FUNCTION_BLOCK FB_System_BelHa
VAR_INPUT
	Freigabe_auto			: BOOL:=TRUE;
	Betrieb_Anford_auto		: BOOL:=TRUE;
	Regelung_Sollw_auto		: REAL;
	AdressType				: E_DALIV2AddrType;
END_VAR
VAR_OUTPUT
	{attribute 'OPC.UA.DA' := '1'}Steuerung				: ST_System_Bel_Steuerung;		
	{attribute 'OPC.UA.DA' := '1'}Stellwert				: ST_System_Bel_Stellwert;		
	{attribute 'OPC.UA.DA' := '1'}Zustand					: ST_System_Bel_Zustand;	
	{attribute 'OPC.UA.DA' := '1'}Parameter				: ST_System_Bel_Parameter;		
	Parameter_Regelung		: ST_Bel_Parameter;
	Parameter_Filter		: ST_Bel_Parameter;
END_VAR
VAR
	Ablaufsteuerung			: FB_System_BelHa_Ablaufsteuerung;
	Zustandscheck			: FB_System_BelHa_Zustandscheck;
	Logik 					: FB_System_BelHa_Logik;
	Sollwertscheck			: FB_System_BelHa_Sollwertscheck;
	Stellwertscheck			: FB_System_BelHa_Stellwertscheck;

	BeleuchtungGruppe1		: FB_Bel;
	BeleuchtungGruppe2		: FB_Bel;

	TasterGruppe1			: FB_Bel_Taster;
	Steuer_Taster			: FB_Bel_Taster_Steuerung;

	Sensor1					: FB_Bel_Lichtsensor;
	Sensor2					: FB_Bel_Lichtsensor;

	Regelung				: FB_System_BelHa_Regelung;
	Filter					: FB_Bel_Filter;

	Zustand_Bel_Gr1			: ST_BEL_Zustand;
	Zustand_Bel_Gr2			: ST_BEL_Zustand;

	In_Regelung_modus		: BOOL;
	Regelung_Modus_auto		: SINT;


	(*Stellwert der Regelung*)
	Stellwert1_Regelung			: REAL := 100;
	Stellwert2_Regelung			: REAL := 100;

	(*OPCUA Variablen*)
	{attribute 'OPC.UA.DA' := '1'}Ein_Aus_OPCUA: BOOL := TRUE;
	{attribute 'OPC.UA.DA' := '1'}Regelung_OPCUA: BOOL;  		
	{attribute 'OPC.UA.DA' := '1'}Beleuchtung_1_OPCUA: REAL;  
	{attribute 'OPC.UA.DA' := '1'}Beleuchtung_2_OPCUA: REAL;  


	EIN_AUS_Schalter	AT %I* : BOOL;


	Flanke: R_TRIG;
END_VAR
VAR // added by the converter: edge detectors and wires of the graphical bodies
    _w1 : ANY;
END_VAR

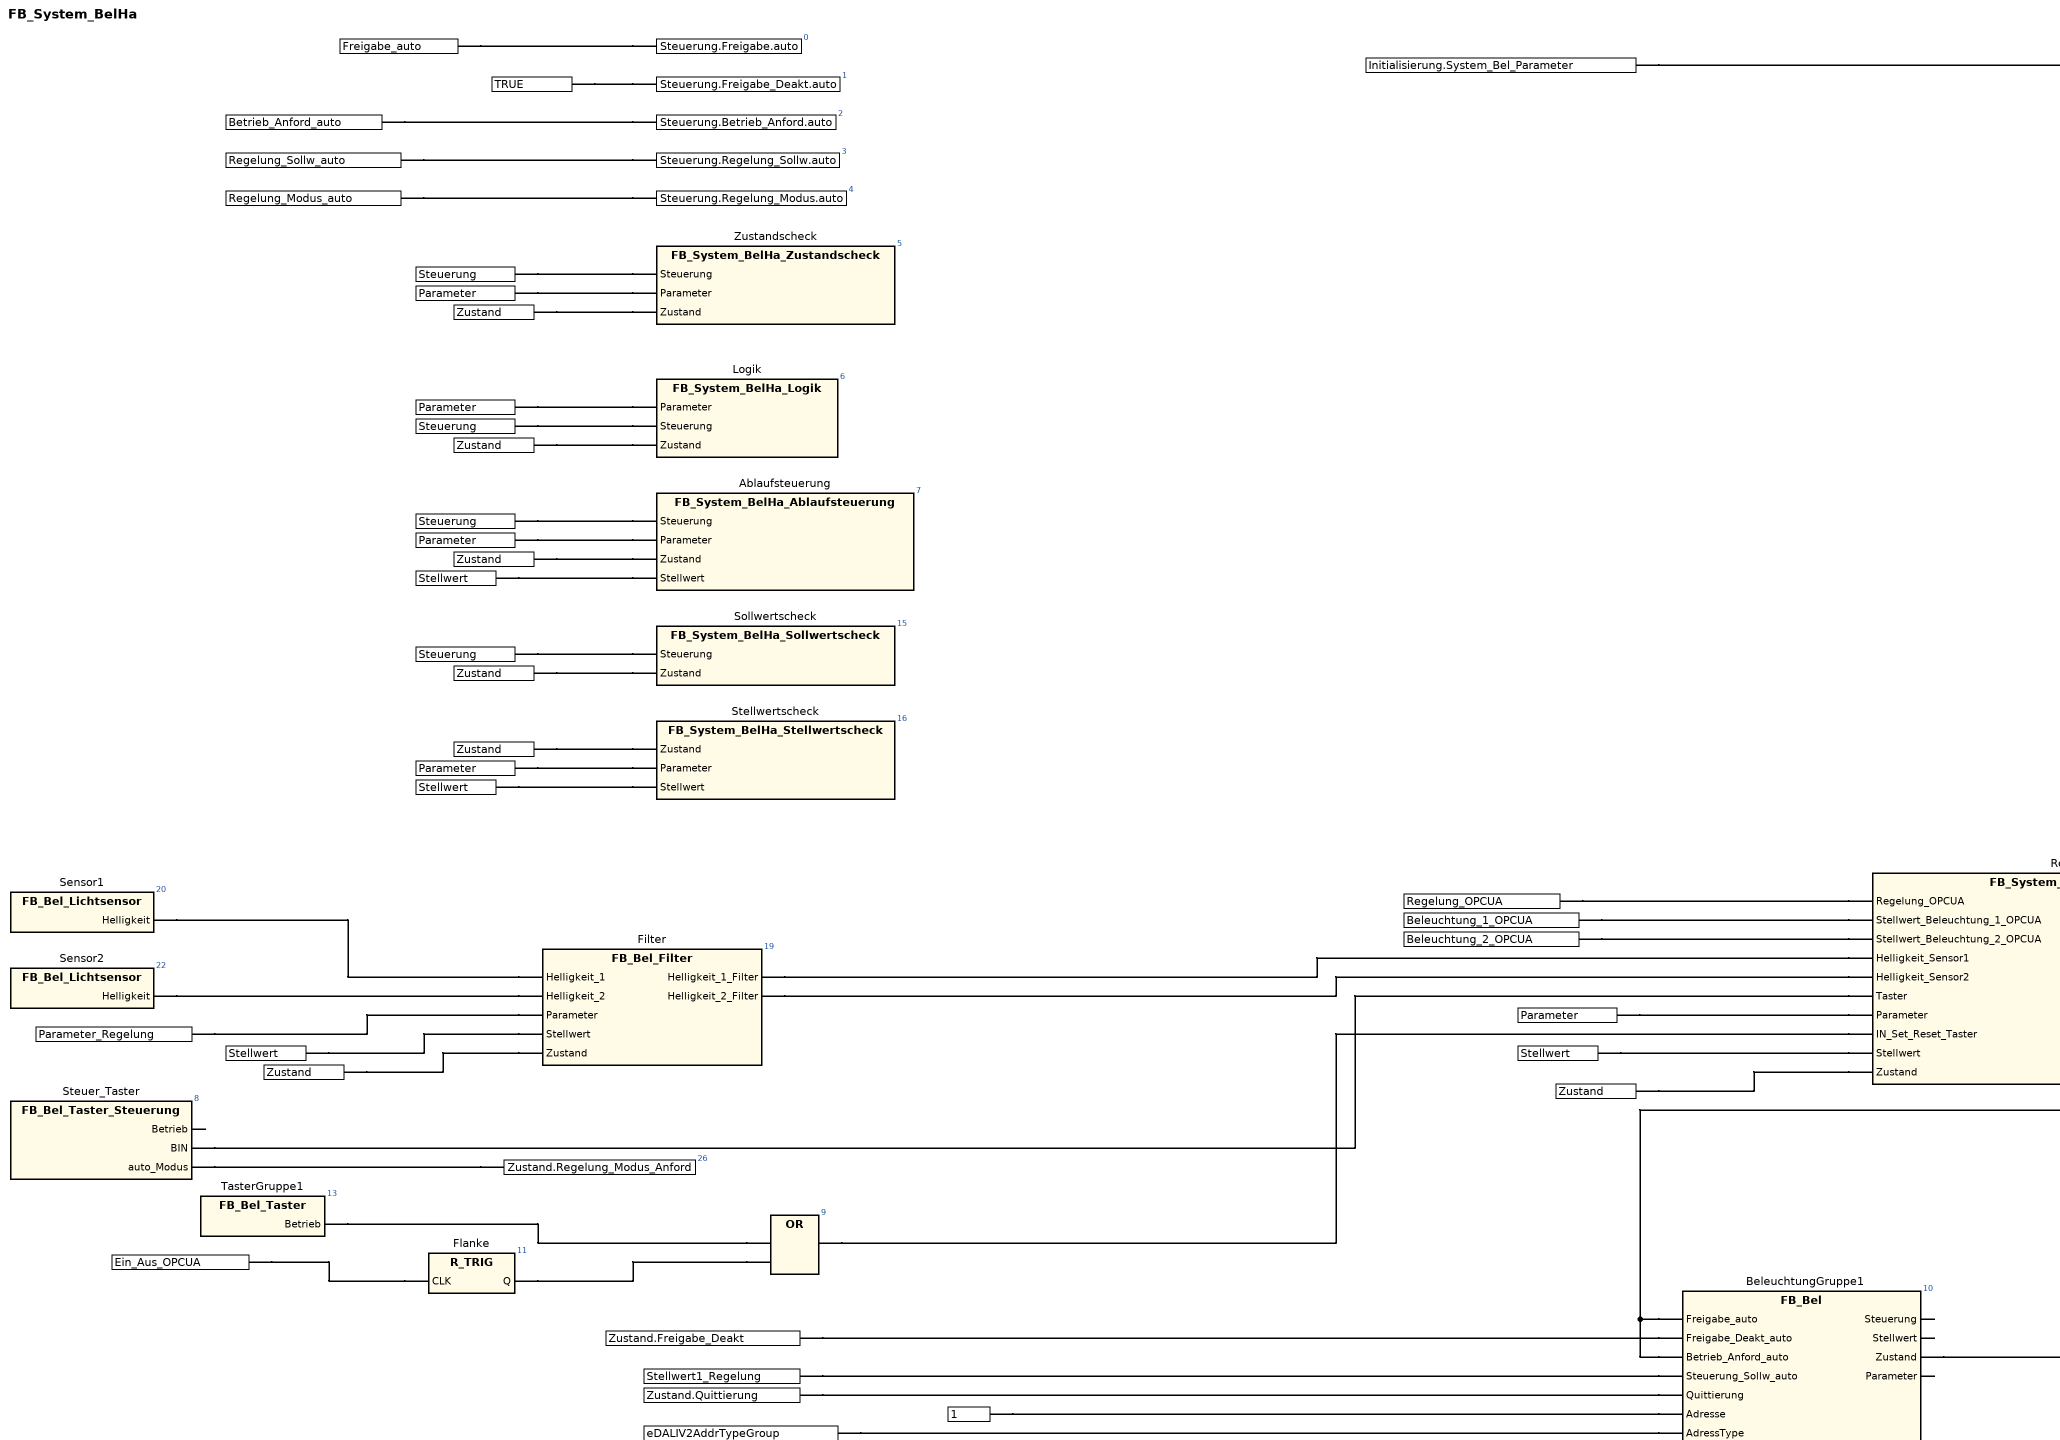
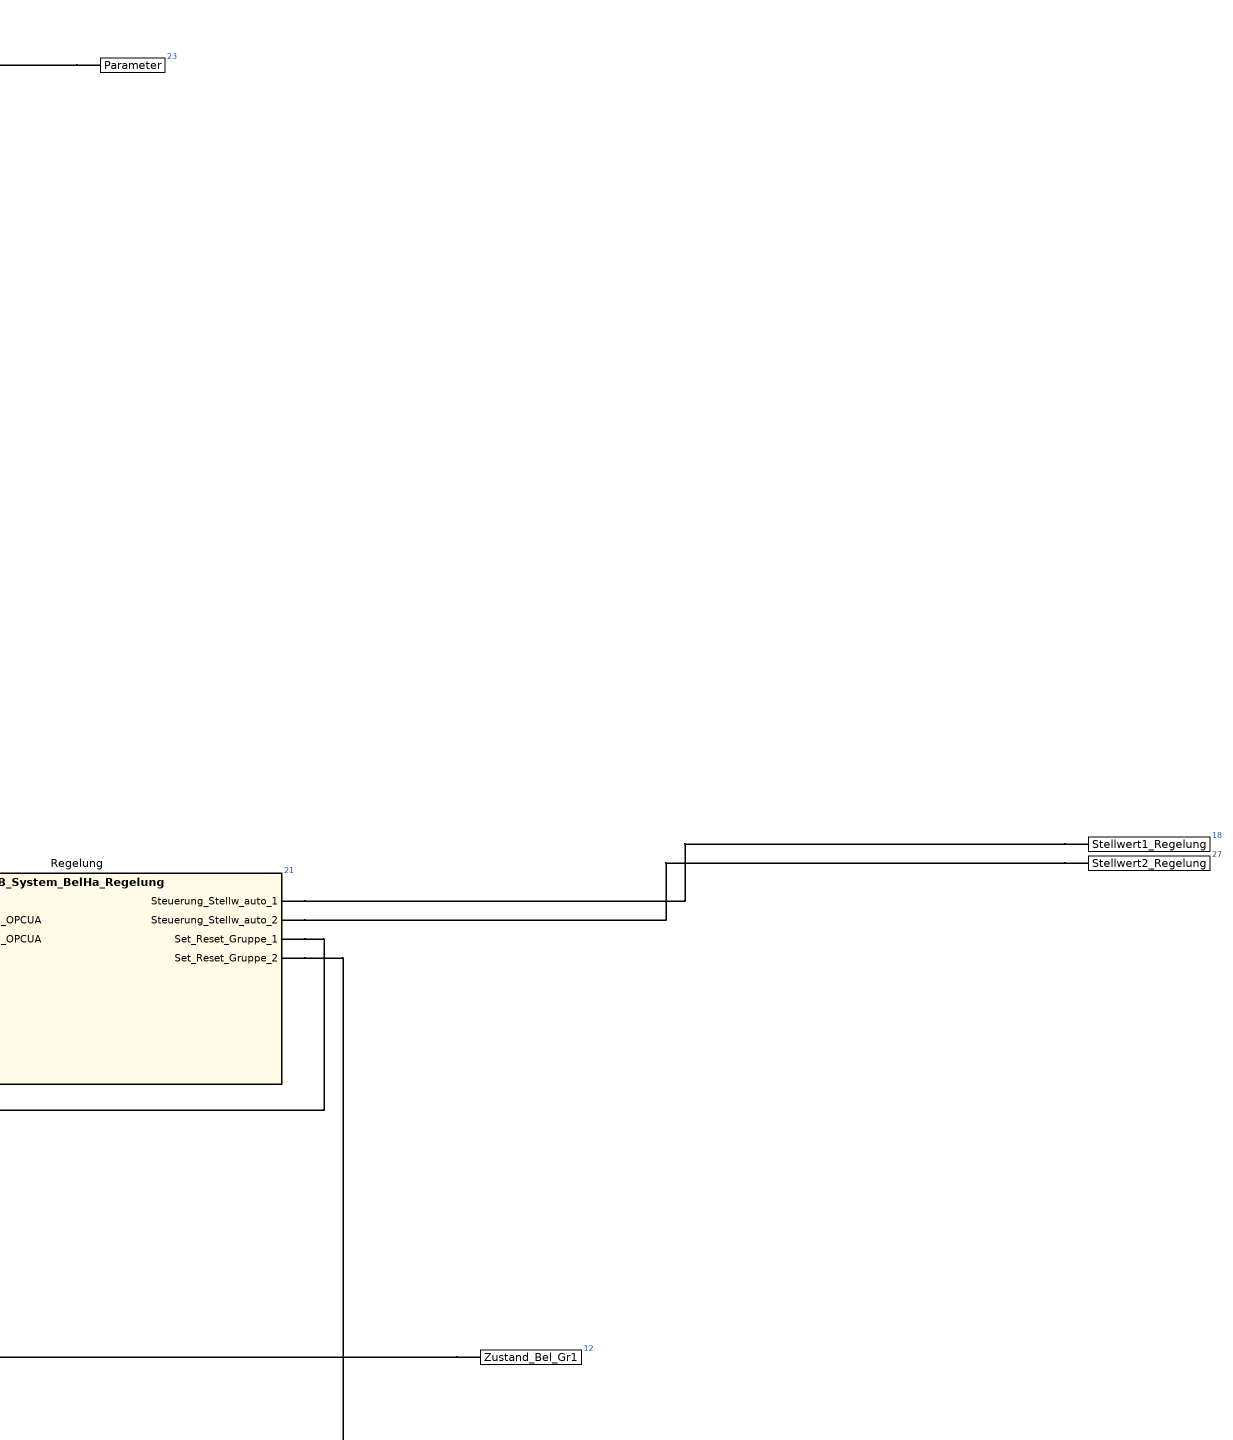
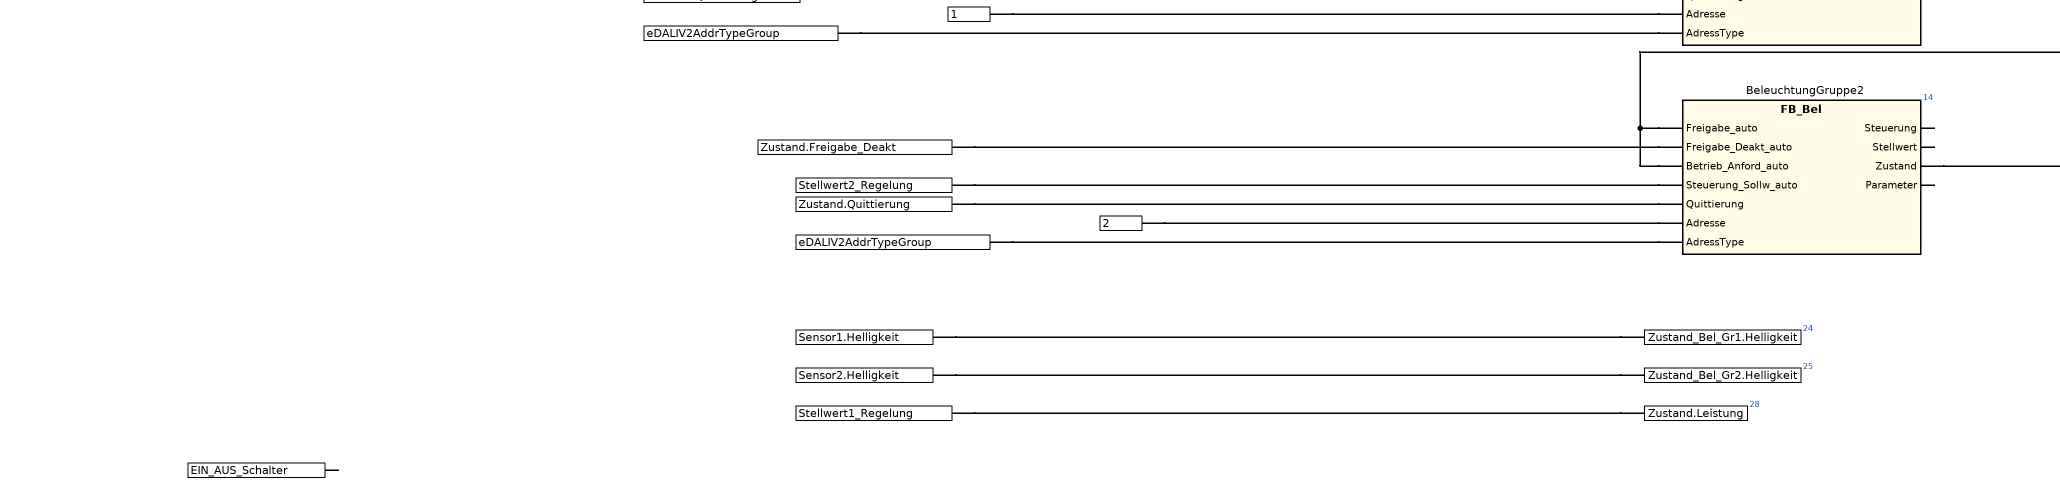
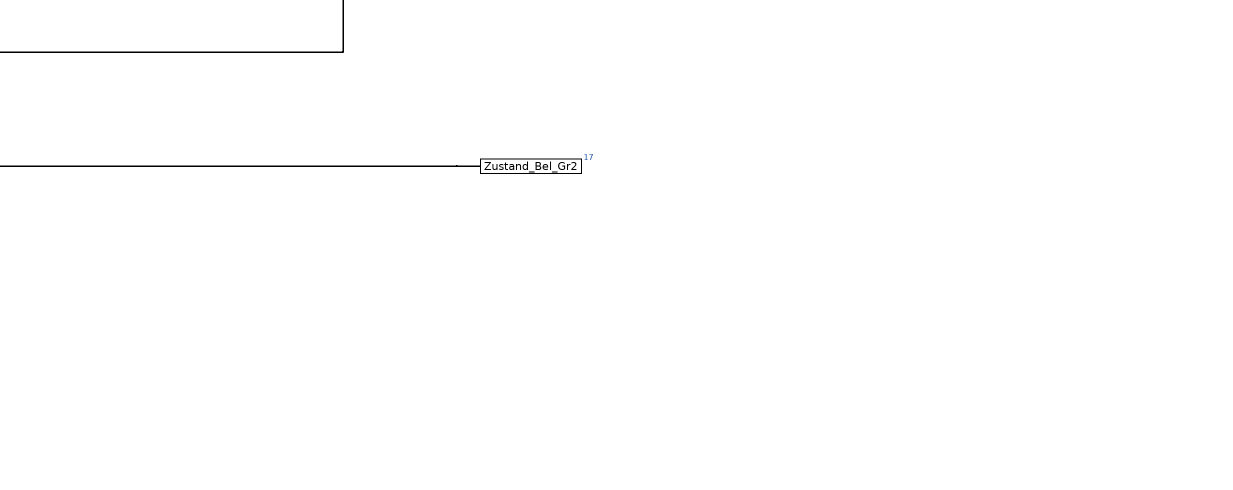
Steuerung.Freigabe.auto := Freigabe_auto;
Steuerung.Freigabe_Deakt.auto := TRUE;
Steuerung.Betrieb_Anford.auto := Betrieb_Anford_auto;
Steuerung.Regelung_Sollw.auto := Regelung_Sollw_auto;
Steuerung.Regelung_Modus.auto := Regelung_Modus_auto;
Zustandscheck(Steuerung := Steuerung, Parameter := Parameter, Zustand := Zustand); // FB_System_BelHa_Zustandscheck
Logik(Parameter := Parameter, Steuerung := Steuerung, Zustand := Zustand); // FB_System_BelHa_Logik
Ablaufsteuerung(Steuerung := Steuerung, Parameter := Parameter, Zustand := Zustand, Stellwert := Stellwert); // FB_System_BelHa_Ablaufsteuerung
Steuer_Taster(); // FB_Bel_Taster_Steuerung
_w1 := TasterGruppe1.Betrieb OR Flanke.Q;
BeleuchtungGruppe1(
    Freigabe_auto := Regelung.Set_Reset_Gruppe_1,
    Freigabe_Deakt_auto := Zustand.Freigabe_Deakt,
    Betrieb_Anford_auto := Regelung.Set_Reset_Gruppe_1,
    Steuerung_Sollw_auto := Stellwert1_Regelung,
    Quittierung := Zustand.Quittierung,
    Adresse := 1,
    AdressType := eDALIV2AddrTypeGroup); // FB_Bel
Flanke(CLK := Ein_Aus_OPCUA); // R_TRIG
Zustand_Bel_Gr1 := BeleuchtungGruppe1.Zustand;
TasterGruppe1(); // FB_Bel_Taster
BeleuchtungGruppe2(
    Freigabe_auto := Regelung.Set_Reset_Gruppe_2,
    Freigabe_Deakt_auto := Zustand.Freigabe_Deakt,
    Betrieb_Anford_auto := Regelung.Set_Reset_Gruppe_2,
    Steuerung_Sollw_auto := Stellwert2_Regelung,
    Quittierung := Zustand.Quittierung,
    Adresse := 2,
    AdressType := eDALIV2AddrTypeGroup); // FB_Bel
Sollwertscheck(Steuerung := Steuerung, Zustand := Zustand); // FB_System_BelHa_Sollwertscheck
Stellwertscheck(Zustand := Zustand, Parameter := Parameter, Stellwert := Stellwert); // FB_System_BelHa_Stellwertscheck
Zustand_Bel_Gr2 := BeleuchtungGruppe2.Zustand;
Stellwert1_Regelung := Regelung.Steuerung_Stellw_auto_1;
Filter(
    Helligkeit_1 := Sensor1.Helligkeit,
    Helligkeit_2 := Sensor2.Helligkeit,
    Parameter := Parameter_Regelung,
    Stellwert := Stellwert,
    Zustand := Zustand); // FB_Bel_Filter
Sensor1(); // FB_Bel_Lichtsensor
Regelung(
    Regelung_OPCUA := Regelung_OPCUA,
    Stellwert_Beleuchtung_1_OPCUA := Beleuchtung_1_OPCUA,
    Stellwert_Beleuchtung_2_OPCUA := Beleuchtung_2_OPCUA,
    Helligkeit_Sensor1 := Filter.Helligkeit_1_Filter,
    Helligkeit_Sensor2 := Filter.Helligkeit_2_Filter,
    Taster := Steuer_Taster.BIN,
    Parameter := Parameter,
    IN_Set_Reset_Taster := _w1,
    Stellwert := Stellwert,
    Zustand := Zustand); // FB_System_BelHa_Regelung
Sensor2(); // FB_Bel_Lichtsensor
Parameter := Initialisierung.System_Bel_Parameter;
Zustand_Bel_Gr1.Helligkeit := Sensor1.Helligkeit;
Zustand_Bel_Gr2.Helligkeit := Sensor2.Helligkeit;
Zustand.Regelung_Modus_Anford := Steuer_Taster.auto_Modus;
Stellwert2_Regelung := Regelung.Steuerung_Stellw_auto_2;
Zustand.Leistung := Stellwert1_Regelung;
// EIN_AUS_Schalter: input not connected

END_FUNCTION_BLOCK

(* stored: Version 1.1.0.1, ProductVersion 3.1.4024.9
   POU FB_System_BelHa: Id {5309ec06-474b-4677-81fb-6cf3831d1c59}, SpecialFunc None *)
